Fanuc KAREL source: kf00101.KL

-- PROVISIONAL review KL for V940-1; original PC SHA256 be942cdcae1483ed6dc5f6b93791545c6430b46836f587b21fc4e68f95070bcc
-- Incomplete behavior may be omitted. Consult companion uncertainty JSON. Do not deploy.
PROGRAM KF00101
%NOLOCKGROUP
BEGIN
  -- V9_ZERO_TABLE_METADATA_HINT layout=0002_ascii; no indexed target words; source/name/runtime held
  -- UNRESOLVED_PC offsets 5-16; opcodes 2E,23
  -- UNRESOLVED_PC offsets 21-32; opcodes 2E,23
  -- UNRESOLVED_PC offsets 37-63; opcodes 27,27,9D,22,27,9D,31,7E,4A
  -- UNRESOLVED_PC offsets 68-72; opcodes 7F
END KF00101
